{attribute addProperty BoxType "EK1300-0000-0017"}
{attribute addProperty Id "Status_UsAT %I*Status_Us_D944C060810Status_UpAT %I*Status_Up_D944C060810WcStateAT %I*WcState_F855686C1620InfoDataAT %I*InfoData_192954DE1620"}
{attribute addProperty CRC "3115393739"}
{attribute addProperty SizeInBites "48"}
{attribute addProperty SizeInBytes "6"}
TYPE EK1300_D787878A :
STRUCT
	{attribute addProperty Name "Status_Us"}
	Status_Us : Status_Us_D944C060;
	{attribute addProperty Name "Status_Up"}
	Status_Up : Status_Up_D944C060;
	{attribute addProperty Name "WcState"}
	WcState : WcState_F855686C;
	{attribute addProperty Name "InfoData"}
	InfoData : InfoData_192954DE;
END_STRUCT
END_TYPE

(* stored: Version 1.2.0.0, ProductVersion 3.1.4024.9
   DUT EK1300_D787878A: Id {5cc9b973-04db-4026-a155-4fe307eaf8cf} *)
